// TIA Portal V17 export
// export: Created 2023-02-26T22:59:53.2159837Z, ExportSetting WithDefaults, DisplayName Totally Integrated Automation Portal, DisplayVersion V17, DisplayName TIA Portal Openness, DisplayVersion V17, DisplayName TIA Portal Version Control Interface, DisplayVersion V17, DisplayName TIA Portal Test Suite Advanced, DisplayVersion V17, DisplayName STEP 7 Professional, DisplayVersion V17, DisplayName SIMATIC Energy Suite, DisplayVersion V17, DisplayName STEP 7 Safety, DisplayVersion V17, DisplayName WinCC Professional, DisplayVersion V17
DATA_BLOCK "LOG_CountPackages_DB_1"   // DB37
VERSION : 0.1
// stored: AutoNumber true, InstanceOfName LOG_CountPackage, InstanceOfType FB
"LOG_CountPackage"
   // VAR_INPUT
   //    StartLine : Bool;
   //    Detector : Bool;
   //    ResetCountButton : Bool;
   // END_VAR
   // VAR_OUTPUT
   //    Quantity : Int;
   // END_VAR
   // VAR RETAIN
   //    IEC_Counter_0_Instance { ExternalAccessible := 'False'; ExternalVisible := 'False'; ExternalWritable := 'False'} : CTU_INT;
   //    N_Detector { S7_SetPoint := 'True'} : Bool;
   // END_VAR
BEGIN
END_DATA_BLOCK
